(* IEC 61131-3 sources: Industry-PLC-LLM/data/PLCBEAD_repo/PLCBEAD_PLCEmbed-main/PLC-BEAD/Source/GEB/GRAY_TO_BYTE, 1 file *)

(* ---- GRAY_TO_BYTE.ST ---- *)
FUNCTION GRAY_TO_BYTE:BYTE

	VAR_INPUT
		IN :	BYTE;
	END_VAR

	GRAY_TO_BYTE := SHR(IN,4) XOR IN;
	GRAY_TO_BYTE := SHR(GRAY_TO_BYTE,2) XOR GRAY_TO_BYTE;
	GRAY_TO_BYTE := SHR(GRAY_TO_BYTE,1) XOR GRAY_TO_BYTE;

END_FUNCTION

PROGRAM program0
  VAR
   	IN :	BYTE;
    LocalOUT  : BYTE;
  END_VAR

  LocalOUT := GRAY_TO_BYTE(IN);
END_PROGRAM
